TYPE ST_GCSpinAxisJogCtrl EXTENDS ST_ServiceCtrlBase:
STRUCT
	Param : ST_GCSpinAxisJogParam;
END_STRUCT
END_TYPE

(* stored: Version 1.1.0.1, ProductVersion 3.1.4026.18
   DUT ST_GCSpinAxisJogCtrl: Id {cff758b5-7948-4ab9-8c9c-40945b180fa4} *)
